(* IEC 61131-3 sources: teller/JD_Teller_LC2_V11/Class/_AlarmX3Para, 1 file *)

(* ---- _AlarmX3Para.st ---- *)
(*!
<Class
	Name               = "_AlarmX3Para"
	Revision           = "0.2"
	RealtimeTask       = "false"
	CyclicTask         = "false"
	BackgroundTask     = "false"
	Sigmatek           = "true"
	OSInterface        = "false"
	HighPriority       = "false"
	Automatic          = "false"
	UpdateMode         = "Prescan"
	SharedCommandTable = "true"
	Objectsize         = "(284,120)">
	<Channels>
		<Server
			Name           = "ClassSvr"
			Initialize     = "false"
			Visualized     = "true"
			WriteProtected = "false">
		</Server>
		<Client Name="Para1" Required="false" Internal="false"/>
		<Client Name="Para2" Required="false" Internal="false"/>
		<Client Name="Para3" Required="false" Internal="false"/>
	</Channels>
	<Network Name="_AlarmX3Para">
		<!-- List of Components in this network -->
		<Components>
			<Object
				Name       = "_base"
				Class      = "_AlarmX0Para"
				Position   = "(270,150)"
				Visualized = "true">
				<Channels>
					<Server Name="ClassSvr"/>
					<Client Name="Acknow"/>
					<Client Name="Config"/>
					<Client Name="Group"/>
				</Channels>
			</Object>
		</Components>
		<Comments>
		</Comments>
		<!-- List of Connections in this network -->
		<Connections>
			<Connection Source="this.ClassSvr" Destination="_base.ClassSvr" Vertices="(742,210),(570,240),"/>
			<Connection Source="_base.Config" Destination="this.Config" Vertices="(270,240),(38,210),"/>
			<Connection Source="_base.Acknow" Destination="this.Acknow" Vertices="(270,300),(38,270),"/>
			<Connection Source="_base.Group" Destination="this.Group" Vertices="(270,360),(38,330),"/>
		</Connections>
		<!-- Headerfiles -->
		<Options>
		</Options>
	</Network>
</Class>
*)
#pragma using _AlarmX0Para

_AlarmX3Para : CLASS
: _AlarmX0Para
  //Servers:
  //Clients:
	Para1 	: CltCh_DINT;
	Para2 	: CltCh_DINT;
	Para3 	: CltCh_DINT;
  //Variables:
  //Functions:

	FUNCTION VIRTUAL GLOBAL GetParaID
		VAR_INPUT
			ppara 	: ^UDINT;
		END_VAR
		VAR_OUTPUT
			retcode 	: UDINT;
		END_VAR;

	FUNCTION VIRTUAL GLOBAL GetParaVal
		VAR_INPUT
			ppara 	: ^DINT;
		END_VAR
		VAR_OUTPUT
			retcode 	: UDINT;
		END_VAR;
  //Tables:
	FUNCTION @STD
		VAR_OUTPUT
			ret_code	: CONFSTATES;
		END_VAR;
	FUNCTION GLOBAL TAB @CT_;
END_CLASS;

//*********************Inserted from .\_AlarmX3Para\_AlarmX3Para_00_00.st*********************

FUNCTION VIRTUAL GLOBAL _AlarmX3Para::GetParaID
  VAR_INPUT
    ppara		: ^UDINT;
  END_VAR
  VAR_OUTPUT
    retcode		: UDINT;
  END_VAR

  retcode := 3;

  if(IsClientConnected(#Para1) = TRUE) then
    ppara^ := (Para1.pCH)$UDINT;
  else
    ppara^ := 0;
  end_if;
  ppara += 4;
  if(IsClientConnected(#Para2) = TRUE) then
    ppara^ := (Para2.pCH)$UDINT;
  else
    ppara^ := 0;
  end_if;
  ppara += 4;
  if(IsClientConnected(#Para3) = TRUE) then
    ppara^ := (Para3.pCH)$UDINT;
  else
    ppara^ := 0;
  end_if;

END_FUNCTION
FUNCTION VIRTUAL GLOBAL _AlarmX3Para::GetParaVal
  VAR_INPUT
    ppara		: ^DINT;
  END_VAR
  VAR_OUTPUT
    retcode		: UDINT;
  END_VAR

  ppara^ := Para1.Read(); ppara += 4;
  ppara^ := Para2.Read(); ppara += 4;
  ppara^ := Para3.Read();

  retcode := 3;

END_FUNCTION
